Yaskawa INFORM job: 1PKT.JBI

/JOB
//NAME 1PKT
//POS
///NPOS 3,3,0,0,0,0
///TOOL 0
///POSTYPE PULSE
///PULSE
C00000=-45679,2023,1827,93032,-31048,-914
C00001=-48702,7109,6199,92969,-28838,-876
C00002=-45679,2023,1827,93032,-31048,-914
BC00000=166789,669556,115787
BC00001=166789,669557,115789
BC00002=166789,669556,115787
//INST
///DATE 2024/08/13 10:14
///ATTR SC,RW
///GROUP1 RB1,BS1
NOP
MOVJ C00000 BC00000 VJ=5.00
MOVL C00001 BC00001 V=25.0  //1
MOVJ C00002 BC00002 VJ=5.00
END
